FUNCTION F_Clear : BOOL //size of data type should not exceed double integer maximum value
VAR_INPUT
	Target: ANY;
END_VAR
VAR
END_VAR

MemSet(
	DestAddr       	:= Target.pValue, 
    FillByte    	:= 0, 
    n   			:= DINT_TO_UDINT(Target.diSize)
);

END_FUNCTION

(* stored: Version 1.1.0.1, ProductVersion 3.1.4024.12
   POU F_Clear: Id {8f6b6663-3989-4b1f-bcad-6655ca3dce55}, SpecialFunc None *)
